// TIA Portal V20 export
DATA_BLOCK "HmiInterface"   // DB197
// stored: Access Published, MemoryReserve 100, Namespace Unit1.Em3
   VAR
      em : "LAF_typeEmInterface";
      emHomedCheck : "Unit1.Em3.typeEmHomedCheck";
      webGuid : "LER_typeSequenceInterface";
   END_VAR
   VAR RETAIN
      cmMasterVirtualAxis : "LBC_typeAxisControlInterface";
      cmUnwinderVirtualAxis : "LBC_typeAxisControlInterface";
      cmDancerRegulatorOnOff : "LBC_typeTwoWayActuatorInterface";
      cmDancerSafetyPinIdlePosition : "LBC_typeDigitalSignalInterface";
      cmLoadCellAnalogInput : "LBC_typeAnalogInputInterface";
      cmDancerEncoderAnalogInput : "LBC_typeAnalogInputInterface";
      cmDancerElectroPneumaticRegulatorAnalogOutput : "LBC_typeAnalogOutputInterface";
      cmWebGuideEpc : "LER_typeCON600Interface";
      cmDancerElectroPneumaticRegulatorSV : LReal;
      cmWebGuideEpc_UnUse : Bool;
   END_VAR
   VAR
      FeedingOneCell : Bool;
      MotionDelayTime : Time;
      JogMode : Bool;
   END_VAR
BEGIN
END_DATA_BLOCK
